(* PLC project Unnamed, Unknown Unnamed 1 *)
(* stored: creationDateTime 2025-12-12T07:30:42, modificationDateTime 2025-12-12T18:30:54 *)

PROGRAM program0
  VAR
    BOTON_ARRANQUE AT %IX100.0 : BOOL;
    BOTON_PARADA AT %IX100.1 : BOOL;
    MOTOR1 AT %QX100.0 : BOOL;
    VALVULA1 AT %QX100.1 : BOOL;
    VALVULA2 AT %QX100.2 : BOOL;
    VALVULA3 AT %QX100.3 : BOOL;
    VALVULA4 AT %QX100.4 : BOOL;
    SENSOR_IR_1 AT %IX100.2 : BOOL;
    SENSOR_IR_2 AT %IX100.3 : BOOL;
    SENSOR_IR_3 AT %IX100.4 : BOOL;
    SENSOR_IR_4 AT %IX100.5 : BOOL;
    SENSOR_PESO_1 AT %IX100.6 : BOOL;
    SENSOR_PESO_2 AT %IX100.7 : BOOL;
  END_VAR
  VAR
    TON0 : TON;
    TON1 : TON;
  END_VAR

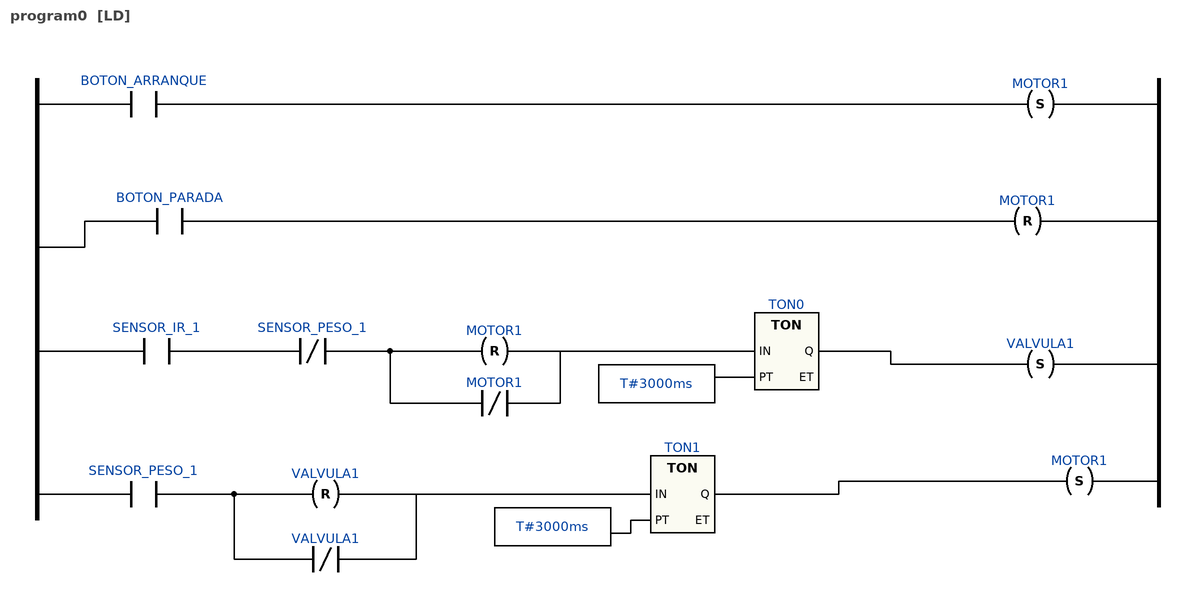
(* LD diagram, written out as Structured Text *)
IF BOTON_ARRANQUE THEN MOTOR1 := TRUE; END_IF;
IF BOTON_PARADA THEN MOTOR1 := FALSE; END_IF;
TON1(IN := SENSOR_PESO_1, PT := T#3000ms);
IF TON1.Q THEN MOTOR1 := TRUE; END_IF;
TON0(IN := SENSOR_IR_1 AND NOT SENSOR_PESO_1, PT := T#3000ms);
IF TON0.Q THEN VALVULA1 := TRUE; END_IF;
IF SENSOR_IR_1 AND NOT SENSOR_PESO_1 THEN MOTOR1 := FALSE; END_IF;
IF SENSOR_PESO_1 THEN VALVULA1 := FALSE; END_IF;
END_PROGRAM

CONFIGURATION Config0
  RESOURCE Res0 ON PLC
    TASK task0(INTERVAL := T#20ms, PRIORITY := 0);
    PROGRAM instance0 WITH task0 : program0;
  END_RESOURCE
END_CONFIGURATION
